FUNCTION_BLOCK Drive_control
VAR_INPUT
	Safety_interlock:BOOL;
	Torque_prediction:INT;
	Speed:INT; (*When this speed is exceeded, the winder will go from torque control to speed control*)
	Movement_detect:BOOL;
	Motor_fed:BOOL;
	Auto_run:BOOL;
	Auto_ref:INT;
	Auto_trail_brakes:BOOL;
	Speed_scale:INT; (*Full lever speed (modified by creep/slow switch*)
	Lh_allowed_speed:INT;
	Rh_allowed_speed:INT;
	Current_limit:INT; (*Current limit in Amps*)
	Max_lever_amps:INT; (*Current ramp rate in Amps*)
	Speed_ramp_rate:INT; (*Speed ramp rate (accel and decel) in mm/s.*)
	Current_ramp_rate:INT; (*Ramp rate of armature current reference in A/s used in torque control*)
	Armature_current:REAL; (*Armature current in Amps*)
	Forward_backout:BOOL;
	Reverse_backout:BOOL;
	Settings_in:dut_Drive_control;
	Mode_in:dut_Mode;
	Brakes_in:dut_Brake;
	Clutch_in:dut_Clutch;
	Power_lever_in:dut_Power_lever;
	Safety_in:dut_Safety;
END_VAR
VAR_OUTPUT
	Enable:BOOL; (*Drive enable signal*)
	Start:BOOL; (*Drive start/run signal*)
	Speed_control:BOOL; (*Drive required to be in speed control*)
	Torque_control:BOOL; (*Drive required to be in torque control*)
	Field_weakening:BOOL; (*Field weakening request (for DC drive)*)
	Brake_release:BOOL;
	Trail_brakes:BOOL;
	Driver_ref_final:INT;
	Speed_ref:INT; (*Speed reference in mm/s*)
	Torque_ref:INT; (*Torque reference in amps*)
	Drive_speed_ref:INT; (*Speed reference to drive scaled according to Speed_10V*)
	Drive_torque_ref:INT; (*Torque reference to drive scaled according to Torque_10V (bipolar)*)
	Combined_ref:INT; (*Speed and torque reference combined output (e.g. for TPD32/DCV104)*)
	No_start:BOOL;
	Stall:BOOL;
	Enable_vs_motor_fed:BOOL;
	hmi_data:dut_hmi_Drive_control;
	Settings_out:dut_Drive_control;
	Mode_out:dut_Mode;
	Brakes_out:dut_Brake;
	Clutch_out:dut_Clutch;
	Power_lever_out:dut_Power_lever;
	Safety_out:dut_Safety;
END_VAR
VAR
	R_TRIG_0: R_TRIG;
	RS_0: RS;
	Torq_ctl_brakes_on: BOOL;
	TON_0: TON;
	Kill_torq_ctl: BOOL;
	RS_1: RS;
	RS_2: RS;
	Lincon_0: Lincon;
	Allowed_speed: INT;
END_VAR
VAR // added by the converter: edge detectors and wires of the graphical bodies
    _w1 : dut_Mode;
    _w2, _w3, _w5, _w6, _w8, _w9, _w10, _w11, _w14, _w15 : BOOL;
    _w4, _w7, _w12, _w16, _w17 : ANY;
    _w13 : INT;
END_VAR

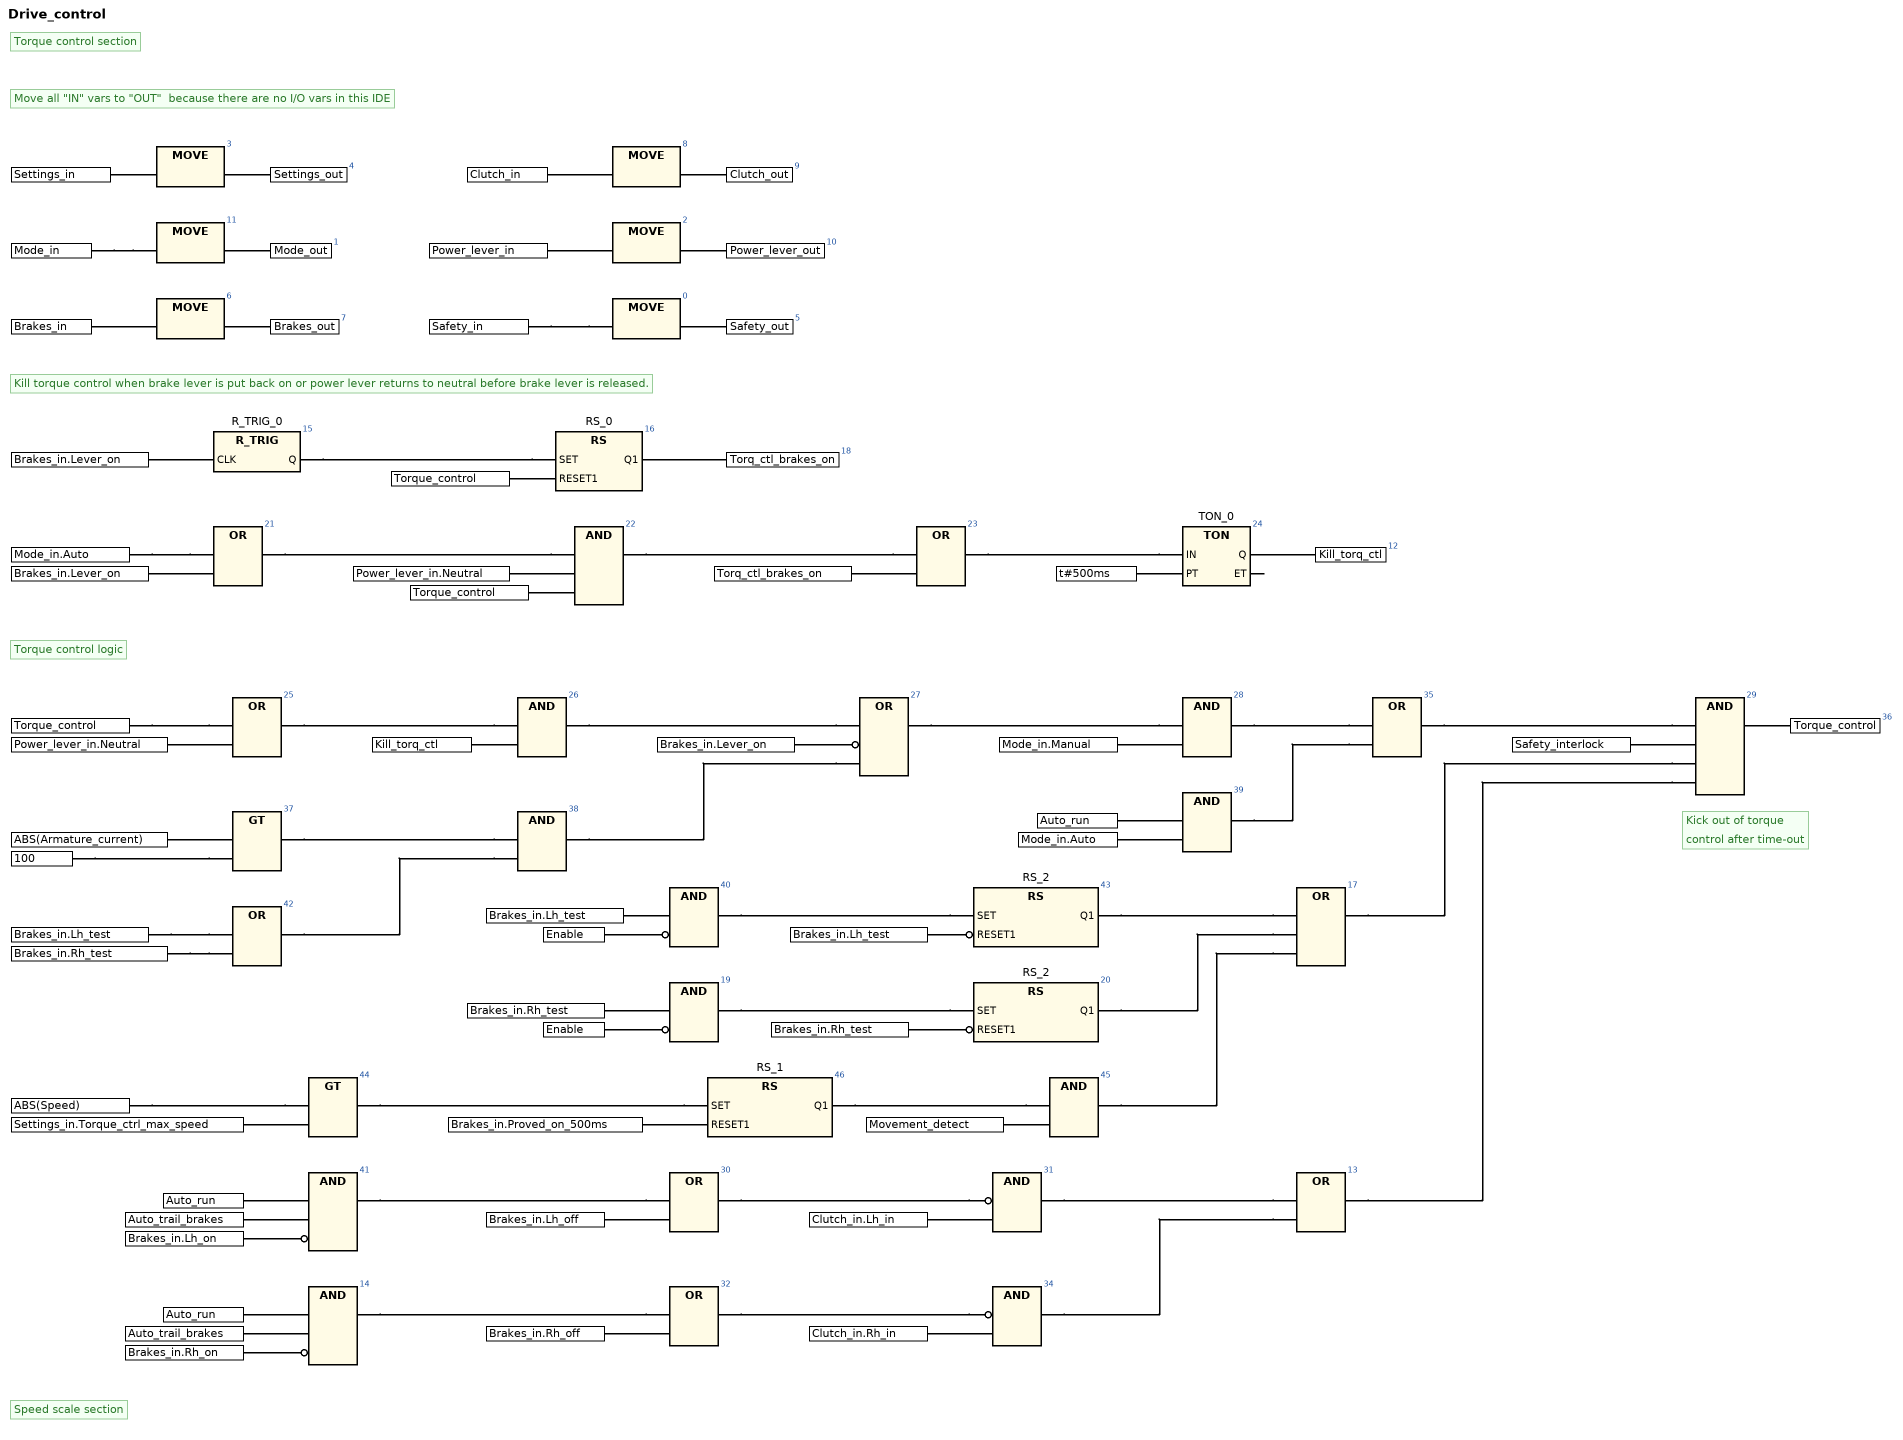
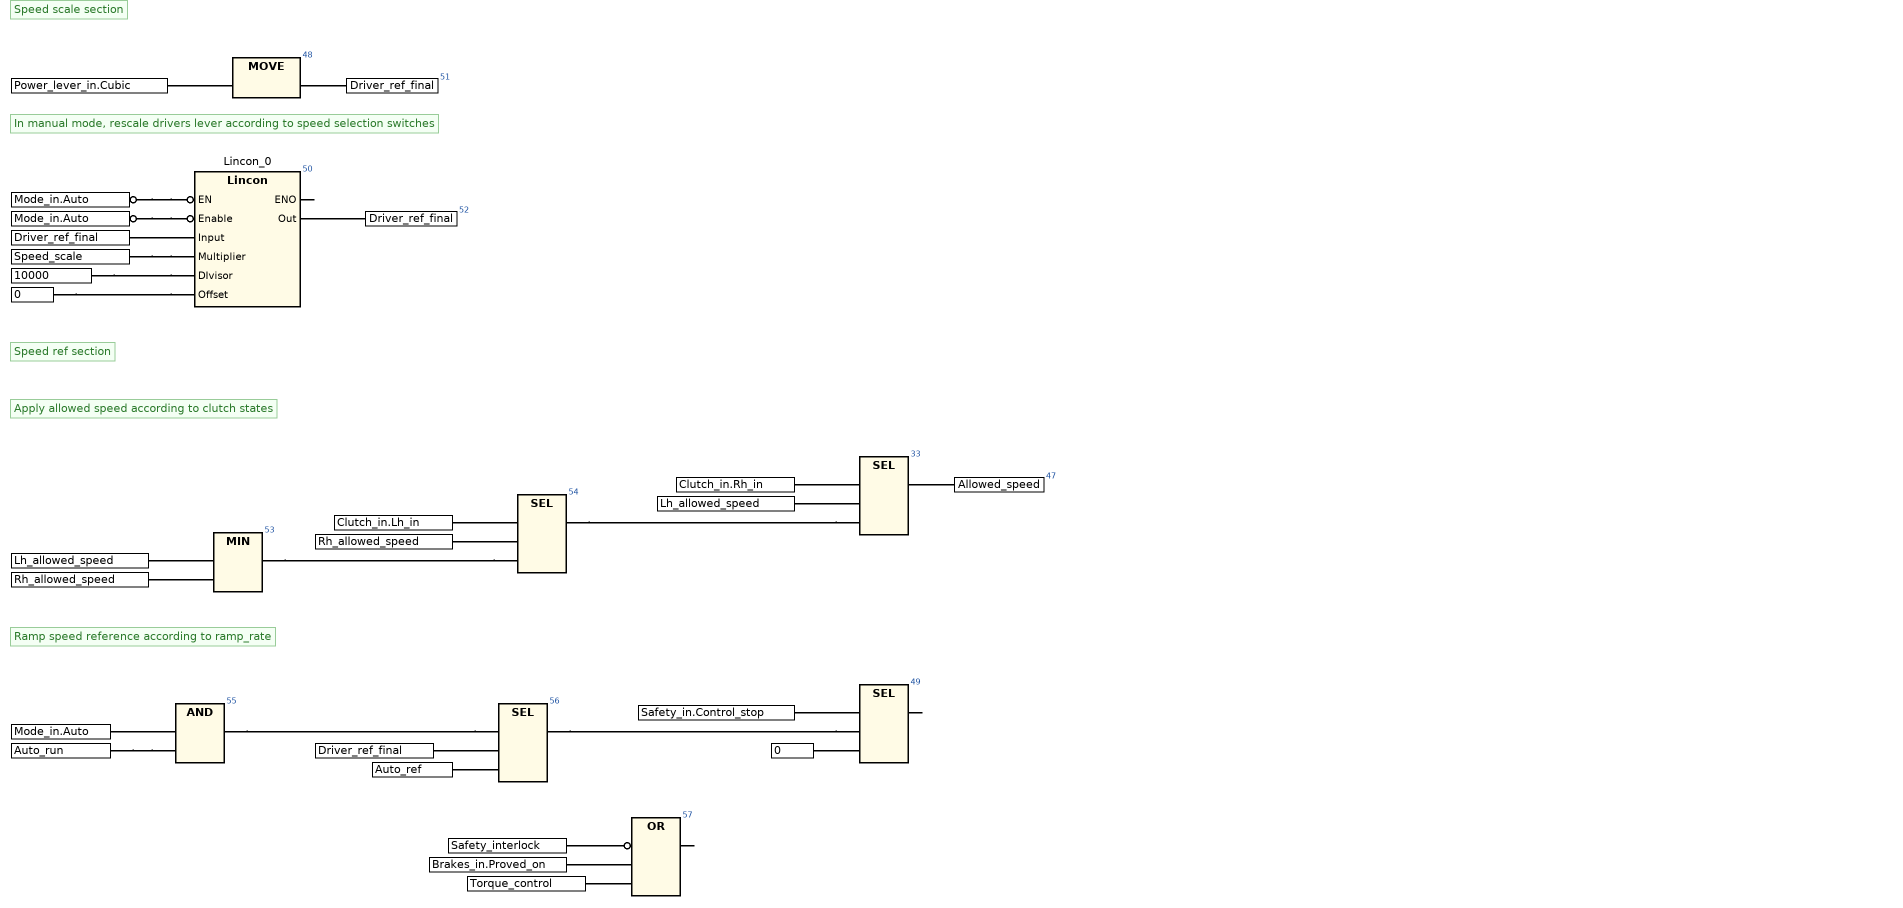
Mode_out := _w1;
// Torque control section
// Move all "IN" vars to "OUT"  because there are no I/O vars in this IDE
Settings_out := Settings_in;
Safety_out := Safety_in;
Brakes_out := Brakes_in;
Clutch_out := Clutch_in;
Power_lever_out := Power_lever_in;
_w1 := Mode_in;
Kill_torq_ctl := TON_0.Q;
_w4 := _w2 OR _w3;
_w5 := Auto_run AND Auto_trail_brakes AND NOT Brakes_in.Rh_on;
// Kill torque control when brake lever is put back on or power lever returns to neutral before brake lever is released.
R_TRIG_0(CLK := Brakes_in.Lever_on); // R_TRIG
RS_0(SET := R_TRIG_0.Q, RESET1 := Torque_control); // RS
// Kick out of torque
// control after time-out
_w7 := RS_2.Q1 OR RS_2.Q1 OR _w6;
Torq_ctl_brakes_on := RS_0.Q1;
RS_2(SET := Brakes_in.Rh_test AND NOT Enable, RESET1 := NOT Brakes_in.Rh_test); // RS
TON_0(IN := (Mode_in.Auto OR Brakes_in.Lever_on) AND Power_lever_in.Neutral AND Torque_control OR Torq_ctl_brakes_on, PT := t#500ms); // TON
// Torque control logic
_w10 := _w9 AND Safety_interlock AND _w7 AND _w4;
_w2 := NOT (_w11 OR Brakes_in.Lh_off) AND Clutch_in.Lh_in;
_w13 := SEL(Clutch_in.Rh_in, Lh_allowed_speed, _w12);
_w3 := NOT (_w5 OR Brakes_in.Rh_off) AND Clutch_in.Rh_in;
_w9 := ((Torque_control OR Power_lever_in.Neutral) AND Kill_torq_ctl OR NOT Brakes_in.Lever_on OR _w8) AND Mode_in.Manual OR _w14;
Torque_control := _w10;
_w8 := (ABS(Armature_current)) > 100 AND _w15;
_w14 := Auto_run AND Mode_in.Auto;
_w11 := Auto_run AND Auto_trail_brakes AND NOT Brakes_in.Lh_on;
_w15 := Brakes_in.Lh_test OR Brakes_in.Rh_test;
RS_2(SET := Brakes_in.Lh_test AND NOT Enable, RESET1 := NOT Brakes_in.Lh_test); // RS
_w6 := RS_1.Q1 AND Movement_detect;
RS_1(SET := (ABS(Speed)) > Settings_in.Torque_ctrl_max_speed, RESET1 := Brakes_in.Proved_on_500ms); // RS
Allowed_speed := _w13;
// Speed scale section
_w16 := Power_lever_in.Cubic;
(* SEL(Safety_in.Control_stop, _w17, 0); result not used *)
// In manual mode, rescale drivers lever according to speed selection switches
IF NOT (NOT Mode_in.Auto) THEN
    Lincon_0(
        Enable := NOT (NOT Mode_in.Auto),
        Input := Driver_ref_final,
        Multiplier := Speed_scale,
        DIvisor := 10000,
        Offset := 0); // Lincon
END_IF
Driver_ref_final := _w16;
Driver_ref_final := Lincon_0.Out;
// Speed ref section
// Apply allowed speed according to clutch states
_w12 := SEL(Clutch_in.Lh_in, Rh_allowed_speed, MIN(Lh_allowed_speed, Rh_allowed_speed));
// Ramp speed reference according to ramp_rate
_w17 := SEL(Mode_in.Auto AND Auto_run, Driver_ref_final, Auto_ref);
(* NOT Safety_interlock OR Brakes_in.Proved_on OR Torque_control; result not used *)

END_FUNCTION_BLOCK

(* stored: Version 1.1.0.1, ProductVersion 3.1.4024.0
   POU Drive_control: Id {20fc2634-4036-4e30-9618-c8d92addbfec}, SpecialFunc None *)
